// TIA Portal V19 export
VAR_GLOBAL   // PLC tag table "LB103"
   LB103_PitTableLoop1_Lp AT %Q113.3 : Bool;   // 317SA1
   LB103_PitTableLoop1_Sel_Down AT %I115.5 : Bool;   // 317SA1
   LB103_PitTableLoop1_Sel_Up AT %I115.4 : Bool;   // 317SA1
END_VAR
